// TwinCAT 3 PLC project Untitled1
// ProgramVersion: 3.1.4026.20
// libraries:
//   Tc2_Standard, * (Beckhoff Automation GmbH)
//   Tc2_System, * (Beckhoff Automation GmbH)
// project tree:
//   / PlcTask.TcTTO
//   POUs/ E_ElevatorState.TcDUT, Elevator.TcPOU, E_PackagingState.TcDUT, FB_TrafficLight.TcPOU, LibrariesAndReusableCode.TcPOU, MachineState.TcDUT, MAIN.TcPOU, Namingconventions.TcPOU, PackagingLine.TcPOU, POU.TcPOU, SpeedCalculation.TcPOU, TankfillingSystem.TcPOU, Thankfillingenum.TcDUT
// real-time tasks:
//   TASK PlcTask: cycle T#10ms, priority 20, ADS port 350

CONFIGURATION Untitled1
    RESOURCE PLC ON TwinCAT3
        TASK PlcTask(INTERVAL := T#10ms, PRIORITY := 20);
        PROGRAM MAIN WITH PlcTask : MAIN;
    END_RESOURCE
END_CONFIGURATION

// ---- POUs/E_ElevatorState.TcDUT
//{attribute 'qualified_only'}
//{attribute 'strict'}
{attribute 'to_string'}
TYPE E_ElevatorState :
(
	//Idle,
    MovingUp,
    MovingDown,
    DoorControl
	//Fault
);
END_TYPE

// ---- POUs/E_PackagingState.TcDUT
//{attribute 'qualified_only'}
//{attribute 'strict'}
{attribute 'to_string'}
TYPE E_PackagingState :
(
	Idle,
    Moving,
    Sealing,
    Error

);
END_TYPE

// ---- POUs/MachineState.TcDUT
//{attribute 'qualified_only'}
{attribute 'strict'}
{attribute 'to_string'}
TYPE MachineState :
(
	off   := 0, 
	on    := 1
	//error := 2
);
END_TYPE

// ---- POUs/Thankfillingenum.TcDUT
//{attribute 'qualified_only'}
//{attribute 'strict'}
{attribute 'to_string'}
TYPE Thankfillingenum :
(
	IDLlE := 0,
	FILLING  := 1,
	FULL  := 2,
	DRAINING  := 3,
	FAULT  := 4
);
END_TYPE

// ---- POUs/MAIN.TcPOU
PROGRAM MAIN
VAR
	LibrariesAndReusableCode :LibrariesAndReusableCode; 
	pou : pou; 
CurrentState : INT; 
Lamp : BOOL; 
variable : BOOL ; 
Elevator : Elevator ; 
PackagingLine :PackagingLine; 
    MainRoad    : FB_TrafficLight;
    SideStreet  : FB_TrafficLight;
	TankfillingSystem:TankfillingSystem; 
END_VAR

 IF CurrentState = 0 THEN 
	Lamp := FALSE; 
ELSIF CurrentState = 1 THEN 
	Lamp := TRUE; 
ELSIF CurrentState = 2 THEN 
	//blink lamp
END_IF

IF variable THEN 
	currentstate := currentstate +1 ; 
	ELSE currentstate := currentstate - 1; 
END_IF

Elevator(); 

POU(); 
LibrariesAndReusableCode(Number := -5);

// Main Road Code Implementation


// Side Street Code Implementation



// Traffic Light Code Implementation

// Main road: long green
MainRoad(
    tRedTime    := T#5s,
    tYellowTime := T#2s,
    tGreenTime  := T#10S
);

// Side street: short green
SideStreet(
    tRedTime    := T#10s,
    tYellowTime := T#2s,
    tGreenTime  := T#5S
);


PackagingLine(); 
TankfillingSystem();

END_PROGRAM

// ---- POUs/LibrariesAndReusableCode.TcPOU
FUNCTION_BLOCK LibrariesAndReusableCode
VAR_INPUT
	Number : REAL;
END_VAR
VAR_OUTPUT
END_VAR
VAR
	 
END_VAR

// absolute value
IF Number < 0 THEN 
	Number := Number*(-1); 
ELSE
	Number := Number ; 
END_IF

Number := ABS(Number);

END_FUNCTION_BLOCK

// ---- POUs/POU.TcPOU
FUNCTION_BLOCK POU
VAR_INPUT
END_VAR
VAR_OUTPUT
END_VAR
VAR
	CurrentState: MachineState;
	Lamp: BOOL;
END_VAR

IF CurrentState = off THEN 
	Lamp := FALSE; 
ELSIF CurrentState = On THEN 
	Lamp := TRUE; 
ELSIF CurrentState = Error THEN 
	//blink lamp
END_IF

END_FUNCTION_BLOCK

// ---- POUs/Elevator.TcPOU
FUNCTION_BLOCK Elevator
VAR_INPUT
END_VAR
VAR_OUTPUT
END_VAR
VAR
	ePreviousState : INT; 
    
  
    tMove          : TON;
    tDoor          : TON;
	bCallFloor0 : BOOL; 
	bSelect0 : BOOL; 
	bCallFloor1 : BOOL; 
	bCallFloor2 : BOOL; 
	bSelect1 : BOOL; 
	bSelect2 : BOOL; 
	iCurrentFloor  : INT := 0;
	iTargetFloor   : INT;
	eState         : E_ElevatorState;
	DoorisOpen : BOOL; 
	berror: BOOL; 
END_VAR


(* 
IF berror THEN
	eState:= fault; 
END_IF
CASE eState OF

    Idle:
        IF bCallFloor0 OR bSelect0 THEN
            iTargetFloor := 0;
			bCallFloor0 :=0;  
			bSelect0 := 0 ; 
        ELSIF bCallFloor1 OR bSelect1 THEN
            iTargetFloor := 1;
			bCallFloor1 :=0;  
			bSelect1 := 0 ; 
        ELSIF bCallFloor2 OR bSelect2 THEN
            iTargetFloor := 2;
			bCallFloor2 :=0;  
			bSelect2 := 0 ; 
        END_IF;

        IF iTargetFloor > iCurrentFloor THEN
            eState := MovingUp;
        ELSIF iTargetFloor < iCurrentFloor THEN
            eState := MovingDown;
        END_IF;

    MovingUp:
	tMove(IN := TRUE, PT := T#5S);
        IF tMove.Q THEN
            iCurrentFloor := iCurrentFloor + 1;
            tMove(IN := FALSE);
        END_IF;
		IF iCurrentFloor = iTargetFloor THEN
		    ePreviousState := eState ; 
            eState := DoorControl; 
        END_IF;

    MovingDown:
        tMove(IN := TRUE, PT := T#5S);
        IF tMove.Q THEN
            iCurrentFloor := iCurrentFloor - 1;
            tMove(IN := FALSE);
        END_IF;
		IF iCurrentFloor = iTargetFloor THEN
		    ePreviousState := eState ; 
            eState := DoorControl;
        END_IF;

    DoorControl:
	(* send command to open door here and wait that the door opens. Write true to the DoorisOpen variable *)
			DoorisOpen := TRUE; 
			IF DoorisOpen THEN 
				tDoor(IN := TRUE, PT := T#5S);
			END_IF
		ePreviousState := eState ; 
        IF tDoor.Q THEN
			DoorisOpen := FALSE; 
            tDoor(IN := FALSE);
            eState := Idle;
        END_IF;
    Fault: 
END_CASE;*)

END_FUNCTION_BLOCK

// ---- POUs/PackagingLine.TcPOU
FUNCTION_BLOCK PackagingLine
VAR_INPUT
END_VAR
VAR_OUTPUT
END_VAR
VAR
	eState : E_PackagingState := Idle;
    bStart, bStop, bError : BOOL;
    bSensor : BOOL;
    iCount : INT := 0;
    tSeal : TON;

END_VAR

IF bStop THEN
	eState := Idle;
	bStart := FALSE; 
END_IF;

IF berror THEN 
	eState := error;
	bStart := FALSE; 
END_IF

CASE eState OF
	
    Idle:
        IF bStart THEN
            eState := Moving;
			bStop := FALSE; 
        END_IF; 
  
    Moving:
        IF bSensor THEN
            eState := Sealing;
		END_IF

    Sealing:
	    tSeal(IN := TRUE, PT := T#3S);
        IF tSeal.Q THEN
            iCount := iCount + 1;
            eState := Moving;
            tSeal(IN := FALSE);
			bSensor:=FALSE; 
        END_IF;
    Error:
	
        // Handle jam or sensor fault
END_CASE;

END_FUNCTION_BLOCK

// ---- POUs/FB_TrafficLight.TcPOU
FUNCTION_BLOCK FB_TrafficLight
VAR_INPUT
    tRedTime    : TIME;   // Red duration
    tYellowTime : TIME;   // Yellow duration
    tGreenTime  : TIME;   // Green duration
END_VAR
VAR_OUTPUT
    actualLight : INT := 0; // light color at the present instant
END_VAR
VAR
	bRed    : BOOL;
    bYellow : BOOL;
    bGreen  : BOOL;
    eState : INT := 0;    // 0=Red, 1=Yellow, 2=Green
    ton    : TON;
END_VAR

CASE eState OF

    0: // RED
		bYellow := FALSE; 
		bGreen  := FALSE;
        bRed    := TRUE;
		actualLight := 0; 
		
        ton(IN := TRUE, PT := tRedTime);
        IF ton.Q THEN
            ton(IN := FALSE);
            eState := 1;
        END_IF

    1: // YELLOW
         
		bGreen  := FALSE;
        bRed    := FALSE;
		bYellow := TRUE;
		actualLight := 1; 
		
        ton(IN := TRUE, PT := tYellowTime);
        IF ton.Q THEN
            ton(IN := FALSE);
            eState := 2;
        END_IF

    2: // GREEN
        bYellow := FALSE; 
		bRed    := FALSE;
		bGreen  := TRUE;
		actualLight := 2; 
        
        ton(IN := TRUE, PT := tGreenTime);
        IF ton.Q THEN
            ton(IN := FALSE);
            eState := 0;
        END_IF

END_CASE

END_FUNCTION_BLOCK

// ---- POUs/TankfillingSystem.TcPOU
FUNCTION_BLOCK TankfillingSystem
VAR_INPUT
END_VAR
VAR_OUTPUT
END_VAR
VAR
	(* Inputs *)
	iState       : Thankfillingenum := IDlLE;
    bStart       : BOOL;
    bStop        : BOOL;
    bLowLevel    : BOOL;
    bHighLevel   : BOOL;
    bResetAlarm  : BOOL;

    (* Outputs *)
    bFillValve   : BOOL;
    bDrainValve  : BOOL;
    bAlarm       : BOOL;

    (* Internal *)
   
END_VAR


(* ===================== *)
(* State Machine Logic   *)
(* ===================== *)

IF bStop THEN
    iState := IDlLE;
	bStart := FALSE;
END_IF;

 IF bLowLevel AND bHighLevel THEN (* Sensor fault *)
            iState := FAULT;
 END_IF

CASE iState OF

    IDlLE: (* IDLE *)
        bFillValve := FALSE;
        bDrainValve := FALSE;
        bAlarm := FALSE;

        IF bStart THEN
                iState := FILLING;
        END_IF

    FILLING: (* FILLING *)
        bFillValve := TRUE;
        bDrainValve := FALSE;

        IF bHighLevel THEN
            bFillValve := FALSE;
            iState := FULL;
        END_IF

       

    FULL: (* FULL *)
        bFillValve := FALSE;
        bDrainValve := FALSE;

        IF NOT bHighLevel THEN
            iState := DRAINING;
        END_IF

    DRAINING: (* DRAINING *)
        bFillValve := FALSE;
        bDrainValve := TRUE;

        IF bLowLevel THEN
            bDrainValve := FALSE;
            iState := IDlLE;
        END_IF

    FAULT: (* FAULT *)
        bFillValve := FALSE;
        bDrainValve := FALSE;
        bAlarm := TRUE;
		
        IF bResetAlarm THEN 
            bAlarm := FALSE;
            iState := IDlLE;
        END_IF

END_CASE;

END_FUNCTION_BLOCK

// ---- POUs/Namingconventions.TcPOU
FUNCTION_BLOCK Namingconventions
VAR_INPUT
END_VAR
VAR_OUTPUT
END_VAR
VAR
    bStartButton : BOOL;
    iCycleCount  : INT;
    rTargetSpeed : REAL;
	
	
END_VAR

VAR
	
	x1                :REAL; 
	
	y2                    : REAL; 
	
	temp                 : REAL; 
	
	CalculateAverageSensorValue                  : ton;  
	
	ConvertFahrenheitTemperatureToCelsius              :Ton; 
	
	LogProductionDataToDatabase             : ton; 
	             iMotorSpeed, rTemperatureSetpoint : REAL; 
				 
				 rTemperatureInCelsius : REAL; 
				 rTemperatureInFahrenheit : REAL; 
				  //bStartButton,
END_VAR



bStartButton             := 1; 

iMotorSpeed               := 1; 

rTemperatureSetpoint          := 1; 

bStartButton     := 1; 

// BAD COMMENT: just repeats the code
rTemperatureInCelsius := (rTemperatureInFahrenheit - 32) * 5 / 9;  // convert Fahrenheit to Celsius


// GOOD COMMENT: EXPLAINS WHY!
// We need the Celsius value because our control logic and sensors work in metric units.
rTemperatureInCelsius := (rTemperatureInFahrenheit - 32) * 5 / 9;

END_FUNCTION_BLOCK

// ---- POUs/SpeedCalculation.TcPOU
FUNCTION_BLOCK SpeedCalculation
VAR_INPUT
END_VAR

VAR_OUTPUT
END_VAR
VAR
rSpeed : REAL; 
rDistance: REAL; 
rTime : REAL; 

bError : BOOL; 
nErrorID : INT; 
sErrorText : STRING; 


END_VAR

VAR RETAIN
    iCounter : INT := 0;
END_VAR


VAR PERSISTENT
    iTotalCycles : INT := 0;
END_VAR




rSpeed := rDistance/rTime; 



IF rTime <> 0 THEN // if rTime is not equal to zero
	rSpeed := rDistance/rTime; 
ELSE 
	// Do not devide by rtime because it is zero
END_IF

END_FUNCTION_BLOCK
